{attribute 'GeneratedUsingTerminal: EM7004-0000-9996'}
{attribute addProperty BoxType "EM7004-0000-9996"}
{attribute addProperty Id "OutputAT %Q*ARRAY[0..15] OF BOOL16"}
{attribute addProperty CRC "1538723034"}
{attribute addProperty Size "16"}
TYPE DO_Outputs_A7E1DFAB EXTENDS OutputBase_10CEE7DE :
STRUCT
	{attribute addProperty Name "Output"}
	Output AT %Q* : ARRAY[0..15] OF BOOL;
END_STRUCT
END_TYPE

(* stored: Version 1.2.0.0, ProductVersion 3.1.4024.11
   DUT DO_Outputs_A7E1DFAB: Id {66cc8a2e-0c87-4a23-9842-fb3da5290571} *)
